{attribute 'GeneratedUsingTerminal: ER1008-0001-0016'}
{attribute addProperty BoxType "ER1008-0001-0016"}
{attribute addProperty Id "WcStateAT %I*BOOL1InputToggleAT %I*BOOL1"}
{attribute addProperty CRC "2425479403"}
{attribute addProperty Size "2"}
TYPE WcState_9091E0EB :
STRUCT
	{attribute addProperty Name "WcState"}
	WcState AT %I* : BOOL;
	{attribute addProperty Name "InputToggle"}
	InputToggle AT %I* : BOOL;
END_STRUCT
END_TYPE

(* stored: Version 1.2.0.0, ProductVersion 3.1.4024.11
   DUT WcState_9091E0EB: Id {27664b59-e66e-4aca-bba5-e68d60910dfc} *)
